METHOD StepDecoded : ZCore.ZString
VAR_INPUT
  stepIndex : INT;
END_VAR
VAR_INST
  _stepIndexDecoded : DrillingStep;
END_VAR
_stepIndexDecoded := stepIndex;
stepDecoded := TO_STRING(_stepIndexDecoded);
END_METHOD

END_FUNCTION_BLOCK

// ---- ZApp/Unit/Drilling/_States/DrillingSequenceAutomatic.TcPOU
FUNCTION_BLOCK DrillingSequenceAutomatic EXTENDS DrillingSequence IMPLEMENTS ZCore.ISequence
VAR
  _step : ZCore.Step(DrillingStep.AutomaticBegin, DrillingStep.AutomaticEnd);
END_VAR

IF NOT Busy THEN
  RETURN;
END_IF

IF OnStart(_step) THEN
  ; // init custom sequence variables here ...
END_IF

IF OnStop() THEN
  RETURN; // external stop was triggered
END_IF

IF OnHalt() THEN
  ; // Halting := TRUE; // Uncomment to acknowledge that the sequence is halting
END_IF

REPEAT
  LogStep();

  CASE _step.Index OF
    (* -------------------------------------------------------------------------------------------------------------------------------- *)
    DrillingStep.AutomaticBegin:
    (* -------------------------------------------------------------------------------------------------------------------------------- *)
      IF _step.OnEntry()
      THEN
        ;
      END_IF

      // Await(obj1:=, nextStep:=DrillingStep.AutomaticEnd);
      _step.SetNext(DrillingStep.AutomaticEnd);
    
    (* -------------------------------------------------------------------------------------------------------------------------------- *)
    DrillingStep.AutomaticEnd:
    (* -------------------------------------------------------------------------------------------------------------------------------- *)
      SetBusy(FALSE);
  
  ELSE
    Abort('sequence contains unhandled step');
  END_CASE
UNTIL _step.IsNotRepeatable() OR_ELSE NOT Busy END_REPEAT

END_FUNCTION_BLOCK

// ---- ZApp/Unit/Drilling/_States/DrillingSequenceStop.TcPOU
FUNCTION_BLOCK DrillingSequenceStop EXTENDS DrillingSequence IMPLEMENTS ZCore.ISequence
VAR
  _step : ZCore.Step(DrillingStep.StopBegin, DrillingStep.StopEnd);
  _timerSim : ZAux.Timer;
END_VAR

IF OnStart(_step) THEN
  ; // init custom sequence variables here ...
END_IF

REPEAT
  LogStep();

  CASE _step.Index OF
    (* -------------------------------------------------------------------------------------------------------------------------------- *)
    DrillingStep.StopBegin:
    (* -------------------------------------------------------------------------------------------------------------------------------- *)
      IF _step.OnEntry()
      THEN
        _timerSim.WaitAsync(5);
			END_IF
      
      Await(_timerSim, nextStep:=DrillingStep.StopEnd);
      // _step.SetNext(index:=DrillingStep.StopEnd);

    (* -------------------------------------------------------------------------------------------------------------------------------- *)
    DrillingStep.StopEnd:
    (* -------------------------------------------------------------------------------------------------------------------------------- *)    
      SetBusy(FALSE);
  
  ELSE
    Abort('sequence contains unhandled step');
  END_CASE
UNTIL _step.IsNotRepeatable() OR_ELSE NOT Busy END_REPEAT

END_FUNCTION_BLOCK

// ---- ZApp/Unit/Drilling/_States/DrillingSequenceGoHome.TcPOU
FUNCTION_BLOCK DrillingSequenceGoHome EXTENDS DrillingSequence IMPLEMENTS ZCore.ISequence
VAR
  _step : ZCore.Step(DrillingStep.GohomeBegin, DrillingStep.GohomeEnd);
  _timer : ZAux.Timer;
END_VAR

IF NOT Busy THEN
  RETURN;
END_IF

IF OnStart(_step) THEN
  ; // init custom sequence variables here ...
END_IF

IF OnStop() THEN
  RETURN; // external stop was triggered
END_IF

IF OnHalt() THEN
  ; // Halting := TRUE; // Uncomment to acknowledge that the sequence is halting
END_IF

REPEAT
  LogStep();

  CASE _step.Index OF
    (* -------------------------------------------------------------------------------------------------------------------------------- *)
    DrillingStep.GoHomeBegin:
    (* -------------------------------------------------------------------------------------------------------------------------------- *)
      IF _step.OnEntry()
      THEN
        _timer.WaitAsync(2);
			END_IF
      
      Await(_timer, nextStep:=DrillingStep.GoHomeEnd);
      // _step.SetNext(index:=DrillingStep.GoHomeEnd);

    (* -------------------------------------------------------------------------------------------------------------------------------- *)
    DrillingStep.GoHomeEnd:
    (* -------------------------------------------------------------------------------------------------------------------------------- *)
      SetBusy(FALSE);
  
  ELSE
    Abort('sequence contains unhandled step');
  END_CASE
UNTIL _step.IsNotRepeatable() OR_ELSE NOT Busy END_REPEAT

END_FUNCTION_BLOCK

// ---- ZApp/Unit/Drilling/_States/DrillingSequenceFaultReaction.TcPOU
FUNCTION_BLOCK DrillingSequenceFaultReaction EXTENDS DrillingSequence IMPLEMENTS ZCore.ISequence
VAR
  _step : ZCore.Step(DrillingStep.FaultReactionBegin, DrillingStep.FaultReactionEnd);
  _timerSim : ZAux.Timer;
END_VAR

IF OnStart(_step) THEN
  ; // init custom sequence variables here ...
END_IF

REPEAT
  LogStep();

  CASE _step.Index OF
    (* -------------------------------------------------------------------------------------------------------------------------------- *)
    DrillingStep.FaultReactionBegin:
    (* -------------------------------------------------------------------------------------------------------------------------------- *)
      IF _step.OnEntry()
      THEN
        _timerSim.WaitAsync(5);
			END_IF
      
      Await(_timerSim, nextStep:=DrillingStep.FaultReactionEnd);
      // _step.SetNext(index:=DrillingStep.FaultReactionEnd);

    (* -------------------------------------------------------------------------------------------------------------------------------- *)
    DrillingStep.FaultReactionEnd:
    (* -------------------------------------------------------------------------------------------------------------------------------- *)    
      SetBusy(FALSE);
  
  ELSE
    Abort('sequence contains unhandled step');
  END_CASE
UNTIL _step.IsNotRepeatable() OR_ELSE NOT Busy END_REPEAT

END_FUNCTION_BLOCK

// ---- ZApp/Unit/Assembly/AssemblyUnit.TcPOU
/// Declaration of a distinct unit of this application
FUNCTION_BLOCK AssemblyUnit EXTENDS ZApplication.Unit IMPLEMENTS IAssembly, ZAux.IStateMachineListener
VAR
  _equipment : AssemblyEquipment(THIS^);
  _data : AssemblyDataRef;
  _com : AssemblyComRef;

  _boot : AssemblySequenceBoot(THIS^);
  _automatic : AssemblySequenceAutomatic(THIS^);
  _stop : AssemblySequenceStop(THIS^);
  _gohome : AssemblySequenceGoHome(THIS^);
  _faultReaction : AssemblySequenceFaultReaction(THIS^);
  
  _statemachine : ZApplication.UnitStateMachine;

  _observeTimer : ZAux.Timer;
END_VAR

{attribute 'ZId' := '23221439-50f6-4bf8-9080-f9c9a764eb63'}

IF _observeTimer.Done THEN
  _observeTimer.WaitAsync(0.1);
  
  // monitor _com for requested actions (e.g. start homing, start automatic mode, ...)
  ObserveRequest(_com.Subscribe.Request.Start, ZApplication.UnitStateMachineState.Automatic);
  ObserveRequest(_com.Subscribe.Request.Stop, ZApplication.UnitStateMachineState.Stop);
  ObserveRequest(_com.Subscribe.Request.GoHome, ZApplication.UnitStateMachineState.GoHome);
  ObserveRequest(_com.Subscribe.Request.Halt, ZApplication.UnitStateMachineState.Halt);
  
  // provide relevant information via ADS
  _com.Publish.Request.Stop := _stateMachine.IsTransitionAllowed(ZApplication.UnitStateMachineState.Stop);
  _com.Publish.Request.Start := _stateMachine.IsTransitionAllowed(ZApplication.UnitStateMachineState.Automatic);
  _com.Publish.Request.GoHome := _stateMachine.IsTransitionAllowed(ZApplication.UnitStateMachineState.GoHome);
  _com.Publish.Request.Halt := _stateMachine.IsTransitionAllowed(ZApplication.UnitStateMachineState.Halt);

  _com.Publish.State := _stateMachine.State();
END_IF

METHOD FB_init : BOOL
VAR_INPUT
  bInitRetains : BOOL; // if TRUE, the retain variables are initialized (warm start / cold start)
  bInCopyCode : BOOL;  // if TRUE, the instance afterwards gets moved into the copy code (online change)
  parent : ZCore.IManagedObject; // caller of the Unit's cyclic method. If the Unit runs in its own context use 0
  name : ZCore.ZString;  // name of this unit as it should show up in the logger
  configdata : REFERENCE TO AssemblyDataConfig;  // reference to the configuration data that is used during boot to configure the Units equipment
  machinedata : REFERENCE TO AssemblyDataMachine; // reference to the machine data that is used through most sequences of the unit (motor speed, axes positions, ...)
  calibrationdata : REFERENCE TO AssemblyDataCalibration;  // reference to calibration that is determined by calibration sequences of the unit (static offsets, shifts)
  com : REFERENCE TO AssemblyCom;  // reference to the communication interface that is used to control this Unit via ADS
END_VAR
_name := name;

// initialize local logger decorator
_loggerDecorator.FB_init(bInitRetains, bInCopyCode, name, ZModuleProgram.Logger);
_alarmingDecorator.FB_init(bInitRetains, bInCopyCode, name, ZModuleProgram.Alarming);

// setup data
_data.Config REF= configdata;
_data.Machine REF= machinedata;
_data.Calibration REF= calibrationdata;
_com.Publish REF= com.Publish;
_com.Subscribe REF= com.Subscribe;

// ------- sequence initialization, map sequences of this unit to the statemachine -------
{attribute '__ZwPlcUnitInitSequenceImplementation__'} // Do not remove this attribute! It is used for code generation.
_statemachine.SetSequence(ZApplication.UnitStateMachineState.Boot, _boot);
_statemachine.SetSequence(ZApplication.UnitStateMachineState.FaultReaction, _faultReaction);
_statemachine.SetSequence(ZApplication.UnitStateMachineState.Gohome, _gohome);
_statemachine.SetSequence(ZApplication.UnitStateMachineState.Stop, _stop);
_statemachine.SetSequence(ZApplication.UnitStateMachineState.Automatic, _automatic);

_statemachine.SetName(_name);
_statemachine.SetListener(THIS^);
_statemachine.SetLogger(_logger);

// set initial state
_statemachine.SetState(ZApplication.UnitStateMachineState.Boot);
_statemachineIntrf := _statemachine;
END_METHOD

/// This method is called by a [Statemachine's startTransition method](xref:ZApplication.UnitStateMachine#startTransition)
/// if a given transition was failed (e.g. the transition is not allowed according to the state diagram of the state machine).
/// The State that was active previously in the StateMachine remains active and `requestedState` indicates which state transition
/// was requested by the user.
METHOD OnStartTransitionFailed
VAR_INPUT
  state : INT;  
  requestedState : INT;
END_VAR
END_METHOD

/// This method is called by a [Statemachine's startTransition method](xref:ZApplication.UnitStateMachine#startTransition)
/// if a given transition was successful. Please note, that at the time this event occurs, `state` still holds the
/// state that was active before calling `startTransition`, there is still one more call to this `state` to allow it to 
/// cleanup.
METHOD OnStartTransitionSucceeded
VAR_INPUT
  state : INT;  
  newState : INT;
END_VAR
END_METHOD

/// This method is called after a transition succeeded, right before the [start method of a sequence](xref:ZAux#start) is called.
/// The parameter `state` indicates the State that is active in the statemachine.
METHOD OnStateEntry
VAR_INPUT
  state : INT;
END_VAR
END_METHOD

/// This method is called after a sequence reported an error, but before the state machine starts its error handling.
METHOD OnStateError
VAR_INPUT
  state : INT;
END_VAR
END_METHOD

/// This method is called after a transition succeeded, right before the [stop method of a sequence](xref:ZAux#start) is called.
/// The parameter `state` indicates the State that is active in the statemachine.
METHOD OnStateExit
VAR_INPUT
  state : INT;  
END_VAR
END_METHOD

/// This method if a State has been executed successfully.
/// The parameter `state` indicates the State that is active in the statemachine.
METHOD OnStateSuccess
VAR_INPUT
  state : INT;    
END_VAR
END_METHOD

END_FUNCTION_BLOCK

// ---- ZApp/Unit/Assembly/_Equipment/AssemblyEquipment.TcPOU
/// This function block is a container for equipment that is used by this unit.
/// Equipment is grouped by its kind (actuator, axes, io, ...).
/// It extends from [ManagedObjectContainer](xref:ZCore.ManagedObjectContainer) such that the parent
/// (= the unit itself) can be passed to equipment instances.
FUNCTION_BLOCK AssemblyEquipment EXTENDS AssemblyContainer
VAR_INPUT
  Io : AssemblyIo(_parent);
  Actuator : AssemblyActuator(_parent);
  Axis : AssemblyAxis(_parent);
  Fieldbus : AssemblyFieldbus(_parent);
  Unit : AssemblyLinkedUnit(_parent);
END_VAR

END_FUNCTION_BLOCK

// ---- ZApp/Unit/Assembly/_SubObjects/AssemblyContainer.TcPOU
FUNCTION_BLOCK AssemblyContainer EXTENDS ZCore.ObjectContainer
VAR_INPUT
END_VAR
VAR_OUTPUT
END_VAR
VAR
  {attribute 'hide'}
  _parent : REFERENCE TO AssemblyUnit;
END_VAR

{ attribute 'hide' }
METHOD FB_init : BOOL
VAR_INPUT
	bInitRetains : BOOL; // if TRUE, the retain variables are initialized (warm start / cold start)
	bInCopyCode : BOOL;  // if TRUE, the instance afterwards gets moved into the copy code (online change)
  unit : REFERENCE TO AssemblyUnit;
END_VAR
_parent REF= unit;
END_METHOD

END_FUNCTION_BLOCK

// ---- ZApp/Unit/Assembly/_Equipment/AssemblyIo.TcPOU
/// This function block is a container for all I/Os that are used by this unit.
/// The parent of all objects can be directly transfered in their constructor (this is only relevant for equipment objects
/// that have to be managed (e.g. [DebouncedInput](xref:ZEquipment.DebouncedInput), [Light](xref:ZEquipment.Light), ...).
FUNCTION_BLOCK AssemblyIo EXTENDS AssemblyContainer
VAR
  {attribute 'hide'}
  _iobridge : ZApplication.IoBridge(_parent);
END_VAR
VAR_INPUT

{region "YellowLight : Light"}
  YellowLight : ZEquipment.Light(_parent);
  {attribute 'ZId' := 'd8b54b94-4c20-4805-9de3-a35aa5023c5d'}
{endregion}

{region "RedLight : Light"}
  RedLight : ZEquipment.Light(_parent);
  {attribute 'ZId' := '810dce14-d302-4e94-b60a-e39841040373'}
{endregion}

{region "GreenLight : Light"}
  GreenLight : ZEquipment.Light(_parent);
  {attribute 'ZId' := 'f5a46fca-074f-4557-8a14-cee504d2eb08'}
{endregion}

{region "PneumaticsOk : DigitalInput"}
  PneumaticsOk : ZEquipment.DigitalInput;
  {attribute 'ZId' := 'e461ecc5-0720-4dc8-ad47-eeb7ce01769f'}
{endregion}

{attribute '__ZwPlcUnitEquipmentDeclaration__'} // Do not remove this attribute! It is used for code generation.
END_VAR

IF _isInitialized
THEN
  RETURN;
END_IF

  _iobridge.SetLogger(_parent._logger);

{region "YellowLight : Light"}
  YellowLight.SetLogger(_parent._logger);
  YellowLight.SetName('YellowLight');
  YellowLight.SetSimulation(on:=_parent._data.Config.Simulated);
  YellowLight.SetLogic(ZEquipment.DigitalLogic.Normal);
  _ioBridge.AddLight(YellowLight, publish := _parent._com.Publish.Equipment.YellowLight, subscribe := _parent._com.Subscribe.Equipment.YellowLight);

  {region "UserInitCode"}
  // put your individual init code for this I/O here
  {endregion}

  {attribute 'ZId' := 'd8b54b94-4c20-4805-9de3-a35aa5023c5d'}
{endregion}

{region "RedLight : Light"}
  RedLight.SetLogger(_parent._logger);
  RedLight.SetName('RedLight');
  RedLight.SetSimulation(on:=_parent._data.Config.Simulated);
  RedLight.SetLogic(ZEquipment.DigitalLogic.Normal);
  _ioBridge.AddLight(RedLight, publish := _parent._com.Publish.Equipment.RedLight, subscribe := _parent._com.Subscribe.Equipment.RedLight);

  {region "UserInitCode"}
  // put your individual init code for this I/O here
  {endregion}

  {attribute 'ZId' := '810dce14-d302-4e94-b60a-e39841040373'}
{endregion}

{region "GreenLight : Light"}
  GreenLight.SetLogger(_parent._logger);
  GreenLight.SetName('GreenLight');
  GreenLight.SetSimulation(on:=_parent._data.Config.Simulated);
  GreenLight.SetLogic(ZEquipment.DigitalLogic.Normal);
  _ioBridge.AddLight(GreenLight, publish := _parent._com.Publish.Equipment.GreenLight, subscribe := _parent._com.Subscribe.Equipment.GreenLight);

  {region "UserInitCode"}
  // put your individual init code for this I/O here
  {endregion}

  {attribute 'ZId' := 'f5a46fca-074f-4557-8a14-cee504d2eb08'}
{endregion}

{region "PneumaticsOk : DigitalInput"}
  PneumaticsOk.SetLogger(_parent._logger);
  PneumaticsOk.SetName('PneumaticsOk');
  PneumaticsOk.SetSimulation(on:=_parent._data.Config.Simulated);
  PneumaticsOk.SetLogic(ZEquipment.DigitalLogic.Normal);
  _ioBridge.AddDigitalInput(PneumaticsOk, publish := _parent._com.Publish.Equipment.PneumaticsOk, subscribe := _parent._com.Subscribe.Equipment.PneumaticsOk);

  {region "UserInitCode"}
  // put your individual init code for this I/O here
  {endregion}

  {attribute 'ZId' := 'e461ecc5-0720-4dc8-ad47-eeb7ce01769f'}
{endregion}

{attribute '__ZwPlcUnitEquipmentImplementation__'} // Do not remove this attribute! It is used for code generation.

_isInitialized := TRUE;

END_FUNCTION_BLOCK

// ---- ZApp/Unit/Assembly/_Equipment/AssemblyActuator.TcPOU
/// This function block is a container for all actuator objects that are used by this unit.
/// The parent of all objects can be directly transfered in their constructor (this is only relevant for equipment objects
/// that have to be managed (e.g. [DebouncedInput](xref:ZEquipment.DebouncedInput), [Light](xref:ZEquipment.Light), ...).
FUNCTION_BLOCK AssemblyActuator EXTENDS AssemblyContainer
VAR
  {attribute 'hide'}
  _actuatorbridge : ZApplication.ActuatorBridge(_parent);
  {attribute 'hide'}
  _iobridge : ZApplication.IoBridge(_parent);
END_VAR
VAR_INPUT

{region "Horizontal : ActuatorDigitalBiLsPlusMinus"}
  Horizontal : AssemblyActuatorHorizontal(_parent);
  {attribute 'ZId' := 'bf04a1fd-9e2a-444c-be25-15a99c5011b8'}
{endregion}

{region "Gripper : ActuatorDigitalMonoPlusLsNo"}
  Gripper : AssemblyActuatorGripper(_parent);
  {attribute 'ZId' := 'd18888e4-9abb-463d-b01d-e5fd8694a677'}
{endregion}

{attribute '__ZwPlcUnitEquipmentDeclaration__'} // Do not remove this attribute! It is used for code generation.

  HorizontalListener : ActuatorHorizontalListener(Horizontal, _parent._equipment.Axis.Vertical, _parent._equipment.Io.YellowLight);
  HorizontalPneumaticsCheckListener : PneumaticsOkActuatorListener(Horizontal, _parent._equipment.Io.PneumaticsOk);
  
  GripperPneumaticsCheckListener : PneumaticsOkActuatorListener(Gripper, _parent._equipment.Io.PneumaticsOk);
END_VAR

IF _isInitialized
THEN
  RETURN;
END_IF

  _actuatorbridge.SetLogger(_parent._logger);

{region "Horizontal : ActuatorDigitalBiLsPlusMinus"}
  Horizontal.SetLogger(_parent._logger);
  Horizontal.SetName(name:='Horizontal', movePlusName:='ToTransport', moveMinusName:='ToAssembly', plusName:='AtTransport', minusName:='AtAssembly');
  Horizontal.SetSimulation(SEL(_parent._data.Config.Simulated, ActuatorDigitalSimulation.Disabled, ZEquipment.ActuatorDigitalSimulation.Automatic));
  Horizontal.SetSimulationUncertainty(uncertainty:=10);
  Horizontal.SetDelay(plusStartDuration:=0, plusEndDuration:=0, minusStartDuration:=0, minusEndDuration:=0, stop:=0);
  Horizontal.SetSwitchDuration(plusDuration:=0.2, minusDuration:=0.2);
  Horizontal.SetMovementDuration(plusDuration:=3, minusDuration:=3);
  Horizontal.SetTimeout(plusDuration:=5, minusDuration:=5);
  _actuatorbridge.AddActuatorDigital(Horizontal, publish := _parent._com.Publish.Equipment.Horizontal, subscribe := _parent._com.Subscribe.Equipment.Horizontal);
  _iobridge.AddDigitalOutput(Horizontal.MinusOutput, publish := _parent._com.Publish.Equipment.HorizontalToAssembly, subscribe := _parent._com.Subscribe.Equipment.HorizontalToAssembly);
  _iobridge.AddDigitalOutput(Horizontal.PlusOutput, publish := _parent._com.Publish.Equipment.HorizontalToTransport, subscribe := _parent._com.Subscribe.Equipment.HorizontalToTransport);
  _iobridge.AddDigitalInput(Horizontal.MinusInput, publish := _parent._com.Publish.Equipment.HorizontalAtAssembly, subscribe := _parent._com.Subscribe.Equipment.HorizontalAtAssembly);
  _iobridge.AddDigitalInput(Horizontal.PlusInput, publish := _parent._com.Publish.Equipment.HorizontalAtTransport, subscribe := _parent._com.Subscribe.Equipment.HorizontalAtTransport);
  {region "UserInitCode"}
  // put your individual init code for this Actuator here
  {endregion}

  {attribute 'ZId' := 'bf04a1fd-9e2a-444c-be25-15a99c5011b8'}
{endregion}

{region "Gripper : ActuatorDigitalMonoPlusLsNo"}
  Gripper.SetLogger(_parent._logger);
  Gripper.SetName(name:='Gripper', movePlusName:='Auf', moveMinusName:='Zu', plusName:='Offen', minusName:='Geschlossen');
  Gripper.SetSimulation(SEL(_parent._data.Config.Simulated, ActuatorDigitalSimulation.Disabled, ZEquipment.ActuatorDigitalSimulation.Automatic));
  Gripper.SetSimulationUncertainty(uncertainty:=10);
  Gripper.SetDelay(plusStartDuration:=0, plusEndDuration:=0, minusStartDuration:=0, minusEndDuration:=0, stop:=0);
  Gripper.SetSwitchDuration(plusDuration:=0, minusDuration:=0);
  Gripper.SetMovementDuration(plusDuration:=1, minusDuration:=1);
  Gripper.SetTimeout(plusDuration:=0, minusDuration:=0);
  _actuatorbridge.AddActuatorDigital(Gripper, publish := _parent._com.Publish.Equipment.Gripper, subscribe := _parent._com.Subscribe.Equipment.Gripper);
  _iobridge.AddDigitalOutput(Gripper.PlusOutput, publish := _parent._com.Publish.Equipment.GripperAuf, subscribe := _parent._com.Subscribe.Equipment.GripperAuf);
  {region "UserInitCode"}
  // put your individual init code for this Actuator here
  {endregion}

  {attribute 'ZId' := 'd18888e4-9abb-463d-b01d-e5fd8694a677'}
{endregion}

{attribute '__ZwPlcUnitEquipmentImplementation__'} // Do not remove this attribute! It is used for code generation.

  HorizontalListener.SetLogger(_parent._logger);
  HorizontalListener.SetName('HorizontalActuatorListener');
  
  HorizontalPneumaticsCheckListener.SetLogger(_parent._logger);
  HorizontalPneumaticsCheckListener.SetName('HorizontalPneumaticsCheckListener');
  HorizontalPneumaticsCheckListener.SetPneumaticsOkIo(_parent._equipment.Io.PneumaticsOk);
  
  GripperPneumaticsCheckListener.SetLogger(_parent._logger);
  GripperPneumaticsCheckListener.SetName('HorizontalPneumaticsCheckListener');
  GripperPneumaticsCheckListener.SetPneumaticsOkIo(_parent._equipment.Io.PneumaticsOk);  

_isInitialized := TRUE;

END_FUNCTION_BLOCK

// ---- ZApp/Unit/Assembly/_Equipment/AssemblyActuatorHorizontal.TcPOU
FUNCTION_BLOCK AssemblyActuatorHorizontal EXTENDS ZEquipment.ActuatorDigitalBiLsPlusMinus

METHOD PUBLIC AtAssembly : BOOL
VAR_INPUT
END_VAR
AtAssembly := IsAtMinus();
END_METHOD

METHOD PUBLIC AtTransport : BOOL
VAR_INPUT
END_VAR
AtTransport := IsAtPlus();
END_METHOD

METHOD PUBLIC ToAssemblyAsync
VAR_INPUT
  startToken : ZCore.IStartToken;
END_VAR
MoveMinusAsync(startToken:=startToken);
END_METHOD

METHOD PUBLIC ToTransportAsync
VAR_INPUT
  startToken : ZCore.IStartToken;
END_VAR
MovePlusAsync(startToken:=startToken);
END_METHOD

END_FUNCTION_BLOCK

// ---- ZApp/Unit/Assembly/_Equipment/AssemblyActuatorGripper.TcPOU
FUNCTION_BLOCK AssemblyActuatorGripper EXTENDS ZEquipment.ActuatorDigitalMonoPlusLsNo

METHOD PUBLIC AufAsync
VAR_INPUT
  startToken : ZCore.IStartToken;
END_VAR
MovePlusAsync(startToken:=startToken);
END_METHOD

METHOD PUBLIC Geschlossen : BOOL
VAR_INPUT
END_VAR
Geschlossen := IsAtMinus();
END_METHOD

METHOD PUBLIC Offen : BOOL
VAR_INPUT
END_VAR
Offen := IsAtPlus();
END_METHOD

METHOD PUBLIC ZuAsync
VAR_INPUT
  startToken : ZCore.IStartToken;
END_VAR
MoveMinusAsync(startToken:=startToken);
END_METHOD

END_FUNCTION_BLOCK

// ---- ZApp/Unit/Assembly/_Equipment/ActuatorHorizontalListener.TcPOU
FUNCTION_BLOCK ActuatorHorizontalListener EXTENDS ZEquipment.ActuatorDigitalMoveListenerSequence
VAR
  _timer : ZAux.Timer;
  _step : ZCore.Step(ActuatorHorizontalListenerStep.PreMoveStepBegin, ActuatorHorizontalListenerStep.PreMoveStepEnd);
  _yellowLight : ZEquipment.ILight;
  _axis : ZEquipment.IAxisFeedbackPosition;
END_VAR

CASE THIS^.Movement
OF
  (* ############################################################################## *)
  ZEquipment.ActuatorDigitalMoveListenerMovementType.PreMoveMinus,
  ZEquipment.ActuatorDigitalMoveListenerMovementType.PreMovePlus:
  (* ############################################################################## *)
    IF OnStart(_step)
    THEN
      ;
    END_IF
    
    REPEAT
      LogStep();
      
      CASE _step.Index OF
        (* -------------------------------------------------------------------------------------------------------------------------------- *)
        ActuatorHorizontalListenerStep.PreMoveStepBegin:
        (* -------------------------------------------------------------------------------------------------------------------------------- *)
          _step.SetNext(ActuatorHorizontalListenerStep.PreMoveStepStartLightBlinking);
    
        (* -------------------------------------------------------------------------------------------------------------------------------- *)
        ActuatorHorizontalListenerStep.PreMoveStepStartLightBlinking:
        (* -------------------------------------------------------------------------------------------------------------------------------- *)
          IF _step.OnEntry()
          THEN
            _logger.Info('Start Light Blinking');
            _yellowLight.Enable(characteristic:=LightCharacteristic.Isophase);
          END_IF
        
          _step.SetNext(ActuatorHorizontalListenerStep.PreMoveStepCheckAxisVerticalPosition);
        
        (* -------------------------------------------------------------------------------------------------------------------------------- *)
        ActuatorHorizontalListenerStep.PreMoveStepCheckAxisVerticalPosition:
        (* -------------------------------------------------------------------------------------------------------------------------------- *)
          IF _step.OnEntry()
          THEN
            _logger.Info('Check Axis Position');
            _timer.WaitAsync(duration:=1.5);
          END_IF
        
          // Check if axis is positioned greater than 5mm
          IF _axis.ActualPosition > 5.0
          THEN
            Abort('Cant Move Actuator, Axis at wrong position, collission may occur');
          ELSE
            Await(obj1:=_timer, nextStep:=ActuatorHorizontalListenerStep.PreMoveStepEnd);
          END_IF          
        
        (* -------------------------------------------------------------------------------------------------------------------------------- *)
        ActuatorHorizontalListenerStep.PreMoveStepEnd:
        (* -------------------------------------------------------------------------------------------------------------------------------- *)
          SetBusy(FALSE);
      
      ELSE
        Abort('sequence contains unhandled step');
      END_CASE
    UNTIL _step.IsNotRepeatable() OR_ELSE NOT Busy END_REPEAT
  
  (* ############################################################################## *)
  ZEquipment.ActuatorDigitalMoveListenerMovementType.PostMoveMinus,
  ZEquipment.ActuatorDigitalMoveListenerMovementType.PostMovePlus:
  (* ############################################################################## *)
    _yellowLight.Enable(characteristic:=LightCharacteristic.FixedOff);
    SetBusy(FALSE);
    
END_CASE

METHOD FB_init : BOOL
VAR_INPUT
 bInitRetains : BOOL;
 bInCopyCode : BOOL;
 actuator : REFERENCE TO ActuatorDigital;
 axis : ZEquipment.IAxisFeedbackPosition;
 light : ZEquipment.ILight;
END_VAR
_yellowLight := light;
_axis := axis;
END_METHOD

END_FUNCTION_BLOCK

// ---- ZApp/Unit/Assembly/_Equipment/PneumaticsOkActuatorListener.TcPOU
FUNCTION_BLOCK PneumaticsOkActuatorListener EXTENDS ZEquipment.ActuatorDigitalMoveListenerSequence
VAR
  _pneumaticsOk : ZEquipment.IDigital;
END_VAR

CASE THIS^.Movement
OF
  ZEquipment.ActuatorDigitalMoveListenerMovementType.PreMoveMinus,
  ZEquipment.ActuatorDigitalMoveListenerMovementType.PreMovePlus:
    // Checking if pneumatics are ok and if not abort actuator action
    IF _pneumaticsOk <> 0 AND_THEN NOT _pneumaticsOk.Enabled
    THEN
      Abort('Pneumatics are not OK; check pressure and try again!');
      RETURN;
		END_IF
    
  ZEquipment.ActuatorDigitalMoveListenerMovementType.PostMoveMinus,
  ZEquipment.ActuatorDigitalMoveListenerMovementType.PostMovePlus:
    ;
    
END_CASE

SetBusy(FALSE);

METHOD FB_init : BOOL
VAR_INPUT
 bInitRetains : BOOL;
 bInCopyCode : BOOL;
 actuator : REFERENCE TO ActuatorDigital;
 pneumaticsOk : ZEquipment.IDigital;
END_VAR
_pneumaticsOk := pneumaticsOk;
END_METHOD

METHOD SetPneumaticsOkIo
VAR_INPUT
  intrf : ZEquipment.IDigital;
END_VAR
_pneumaticsOk := intrf;
END_METHOD

END_FUNCTION_BLOCK

// ---- ZApp/Unit/Assembly/_Equipment/AssemblyAxis.TcPOU
/// This function block is a container for all axis objects that are used by this unit.
/// The parent of all objects can be directly transfered in their constructor (this is only relevant for equipment objects
/// that have to be managed (e.g. [DebouncedInput](xref:ZEquipment.DebouncedInput), [Light](xref:ZEquipment.Light), ...).
FUNCTION_BLOCK AssemblyAxis EXTENDS AssemblyContainer
VAR
  {attribute 'hide'}
  _axisbridge : ZApplication.AxisBridge(_parent);
END_VAR
VAR_INPUT

{region "Vertical : AxisPlcOpenMc"}
  Vertical : ZEquipment.AxisPlcOpenMc(_parent);
  {attribute 'ZId' := '59ce020b-a4f8-4d7a-a0dc-8b778ee4fde8'}
{endregion}

{attribute '__ZwPlcUnitEquipmentDeclaration__'} // Do not remove this attribute! It is used for code generation.
END_VAR

IF _isInitialized
THEN
  RETURN;
END_IF

  _axisbridge.SetLogger(_parent._logger);

{region "Vertical : AxisPlcOpenMc"}
  Vertical.SetLogger(_parent._logger);
  Vertical.SetName(name:='Vertical');
  Vertical.SetSimulation(_parent._data.Config.Simulated);
  _axisbridge.AddAxisPlcOpenMc(axis:=Vertical, publish:=_parent._com.Publish.Equipment.Vertical, subscribe:=_parent._com.Subscribe.Equipment.Vertical);

  {region "UserInitCode"}
  // put your individual init code for this Axis here
  {endregion}

  {attribute 'ZId' := '59ce020b-a4f8-4d7a-a0dc-8b778ee4fde8'}
{endregion}

{attribute '__ZwPlcUnitEquipmentImplementation__'} // Do not remove this attribute! It is used for code generation.

_isInitialized := TRUE;

END_FUNCTION_BLOCK

// ---- ZApp/Unit/Assembly/_Equipment/AssemblyFieldbus.TcPOU
/// This function block is a container for all axis objects that are used by this unit.
/// The parent of all objects can be directly transfered in their constructor (this is only relevant for equipment objects
/// that have to be managed (e.g. [DebouncedInput](xref:ZEquipment.DebouncedInput), [Light](xref:ZEquipment.Light), ...).
FUNCTION_BLOCK AssemblyFieldbus EXTENDS AssemblyContainer
VAR
END_VAR
VAR_INPUT

{attribute '__ZwPlcUnitEquipmentDeclaration__'} // Do not remove this attribute! It is used for code generation.
END_VAR

IF _isInitialized
THEN
  RETURN;
END_IF

{attribute '__ZwPlcUnitEquipmentImplementation__'} // Do not remove this attribute! It is used for code generation.

_isInitialized := TRUE;

END_FUNCTION_BLOCK

// ---- ZApp/Unit/Assembly/_Equipment/AssemblyLinkedUnit.TcPOU
/// This function block is a container for all linked units that are used by this unit.
/// Linked units can be addressed through their individual interface.
FUNCTION_BLOCK AssemblyLinkedUnit EXTENDS AssemblyContainer
VAR_INPUT

{attribute '__ZwPlcUnitEquipmentDeclaration__'} // Do not remove this attribute! It is used for code generation.
END_VAR

IF _isInitialized
THEN
  RETURN;
END_IF

{attribute '__ZwPlcUnitEquipmentImplementation__'} // Do not remove this attribute! It is used for code generation.

_isInitialized := TRUE;

END_FUNCTION_BLOCK

// ---- ZApp/Unit/Assembly/_States/AssemblySequenceBoot.TcPOU
FUNCTION_BLOCK AssemblySequenceBoot EXTENDS AssemblySequence IMPLEMENTS ZCore.ISequence
VAR
  _step : ZCore.Step(AssemblyStep.BootBegin, AssemblyStep.BootEnd);
END_VAR

IF OnStart(_step) THEN
  ; // init custom sequence variables here ...
END_IF

REPEAT
  LogStep();

  CASE _step.Index OF
    (* -------------------------------------------------------------------------------------------------------------------------------- *)
    AssemblyStep.BootBegin:
    (* -------------------------------------------------------------------------------------------------------------------------------- *)
      IF _step.OnEntry()
      THEN
        // initialize equipment
        _io();
        _actuator();
        _fieldbus();
        _axis();
        _unit();
      END_IF
      
      _parent._objectManager.Cyclic();      
      Assert(_parent._objectManager);
      IF _parent._objectManager.Done
      THEN
        _step.SetNext(AssemblyStep.BootSwitchOnPneumaticsOkInSimulation);
      END_IF

    (* -------------------------------------------------------------------------------------------------------------------------------- *)
    AssemblyStep.BootSwitchOnPneumaticsOkInSimulation:
    (* -------------------------------------------------------------------------------------------------------------------------------- *)
      IF _step.OnEntry()
      THEN        
        // This IO is an input so this line will only have some effect if PneumaticsOk is simulated to feedback a 
        // functioning pneumatics system to the application in simulation mode
        _io.PneumaticsOk.Enable(TRUE);
      END_IF
      
      _step.SetNext(index:=AssemblyStep.BootEnd);

    (* -------------------------------------------------------------------------------------------------------------------------------- *)
    AssemblyStep.BootEnd:
    (* -------------------------------------------------------------------------------------------------------------------------------- *)
      SetBusy(FALSE);
      
  ELSE
    Abort('sequence contains unhandled step');
  END_CASE
UNTIL _step.IsNotRepeatable() OR_ELSE NOT Busy END_REPEAT

END_FUNCTION_BLOCK

// ---- ZApp/Unit/Assembly/_SubObjects/AssemblySequence.TcPOU
FUNCTION_BLOCK AssemblySequence EXTENDS ZApplication.Sequence
VAR
  {attribute 'hide'}
  _parent : REFERENCE TO AssemblyUnit;
  _io : REFERENCE TO AssemblyIo;
  _actuator : REFERENCE TO AssemblyActuator;
  _fieldbus : REFERENCE TO AssemblyFieldbus;
  _axis : REFERENCE TO AssemblyAxis;
  _data : REFERENCE TO AssemblyDataRef;
  _unit : REFERENCE TO AssemblyLinkedUnit;  
END_VAR

METHOD FB_init : BOOL
VAR_INPUT
  bInitRetains : BOOL; // if TRUE, the retain variables are initialized (warm start / cold start)
  bInCopyCode : BOOL;  // if TRUE, the instance afterwards gets moved into the copy code (online change)
  unit : REFERENCE TO AssemblyUnit;
END_VAR
_parent REF= unit;
_alarming := unit._alarming;
_io REF= unit._equipment.Io;
_actuator REF= unit._equipment.Actuator;
_fieldbus REF= unit._equipment.Fieldbus;
_axis REF= unit._equipment.Axis;
_unit REF= unit._equipment.Unit;
_data REF= unit._data;
_loggerDiagnostics.SetLogger(unit._logger);
END_METHOD

METHOD StepDecoded : ZCore.ZString
VAR_INPUT
  stepIndex : INT;
END_VAR
VAR_INST
  _stepIndexDecoded : AssemblyStep;
END_VAR
_stepIndexDecoded := stepIndex;
stepDecoded := TO_STRING(_stepIndexDecoded);
END_METHOD

END_FUNCTION_BLOCK

// ---- ZApp/Unit/Assembly/_States/AssemblySequenceAutomatic.TcPOU
FUNCTION_BLOCK AssemblySequenceAutomatic EXTENDS AssemblySequence IMPLEMENTS ZCore.ISequence
VAR
  _step : ZCore.Step(AssemblyStep.AutomaticBegin, AssemblyStep.AutomaticEnd);
END_VAR

IF NOT Busy THEN
  RETURN;
END_IF

IF OnStart(_step) THEN
  ; // init custom sequence variables here ...
END_IF

IF OnStop() THEN
  RETURN; // external stop was triggered
END_IF

IF OnHalt() THEN
  ; // Halting := TRUE; // Uncomment to acknowledge that the sequence is halting
END_IF

REPEAT
  LogStep();

  CASE _step.Index OF
    (* -------------------------------------------------------------------------------------------------------------------------------- *)
    AssemblyStep.AutomaticBegin:
    (* -------------------------------------------------------------------------------------------------------------------------------- *)
      IF _step.OnEntry()
      THEN
        ;
      END_IF

      // Await(obj1:=, nextStep:=AssemblyStep.AutomaticEnd);
      _step.SetNext(AssemblyStep.AutomaticEnd);
    
    (* -------------------------------------------------------------------------------------------------------------------------------- *)
    AssemblyStep.AutomaticEnd:
    (* -------------------------------------------------------------------------------------------------------------------------------- *)
      SetBusy(FALSE);
  
  ELSE
    Abort('sequence contains unhandled step');
  END_CASE
UNTIL _step.IsNotRepeatable() OR_ELSE NOT Busy END_REPEAT

END_FUNCTION_BLOCK

// ---- ZApp/Unit/Assembly/_States/AssemblySequenceStop.TcPOU
FUNCTION_BLOCK AssemblySequenceStop EXTENDS AssemblySequence IMPLEMENTS ZCore.ISequence
VAR
  _step : ZCore.Step(AssemblyStep.StopBegin, AssemblyStep.StopEnd);
  _timerSim : ZAux.Timer;
END_VAR

IF OnStart(_step) THEN
  ; // init custom sequence variables here ...
END_IF

REPEAT
  LogStep();

  CASE _step.Index OF
    (* -------------------------------------------------------------------------------------------------------------------------------- *)
    AssemblyStep.StopBegin:
    (* -------------------------------------------------------------------------------------------------------------------------------- *)
      IF _step.OnEntry()
      THEN
        _timerSim.WaitAsync(5);
			END_IF
      
      Await(_timerSim, nextStep:=AssemblyStep.StopEnd);
      // _step.SetNext(index:=AssemblyStep.StopEnd);

    (* -------------------------------------------------------------------------------------------------------------------------------- *)
    AssemblyStep.StopEnd:
    (* -------------------------------------------------------------------------------------------------------------------------------- *)    
      SetBusy(FALSE);
  
  ELSE
    Abort('sequence contains unhandled step');
  END_CASE
UNTIL _step.IsNotRepeatable() OR_ELSE NOT Busy END_REPEAT

END_FUNCTION_BLOCK

// ---- ZApp/Unit/Assembly/_States/AssemblySequenceGoHome.TcPOU
FUNCTION_BLOCK AssemblySequenceGoHome EXTENDS AssemblySequence IMPLEMENTS ZCore.ISequence
VAR
  _step : ZCore.Step(AssemblyStep.GohomeBegin, AssemblyStep.GohomeEnd);
  _timer : ZAux.Timer;
END_VAR

IF NOT Busy THEN
  RETURN;
END_IF

IF OnStart(_step) THEN
  ; // init custom sequence variables here ...
END_IF

IF OnStop() THEN
  RETURN; // external stop was triggered
END_IF

IF OnHalt() THEN
  ; // Halting := TRUE; // Uncomment to acknowledge that the sequence is halting
END_IF

REPEAT
  LogStep();

  CASE _step.Index OF
    (* -------------------------------------------------------------------------------------------------------------------------------- *)
    AssemblyStep.GoHomeBegin:
    (* -------------------------------------------------------------------------------------------------------------------------------- *)
      IF _step.OnEntry()
      THEN
        _timer.WaitAsync(2);
			END_IF
      
      Await(_timer, nextStep:=AssemblyStep.GoHomeGoToHomePos);
      // _step.SetNext(index:=AssemblyStep.GoHomeEnd);

    (* -------------------------------------------------------------------------------------------------------------------------------- *)
    AssemblyStep.GoHomeGoToHomePos:
    (* -------------------------------------------------------------------------------------------------------------------------------- *)
      IF _step.OnEntry()
      THEN        
        _axis.Vertical.MoveAbsoluteAsync(THIS^, 10.0, 2.0);
      END_IF
      
      Await(obj1:=_axis.Vertical, nextStep:=AssemblyStep.GoHomeEnd);

    (* -------------------------------------------------------------------------------------------------------------------------------- *)
    AssemblyStep.GoHomeEnd:
    (* -------------------------------------------------------------------------------------------------------------------------------- *)
      SetBusy(FALSE);
  
  ELSE
    Abort('sequence contains unhandled step');
  END_CASE
UNTIL _step.IsNotRepeatable() OR_ELSE NOT Busy END_REPEAT

END_FUNCTION_BLOCK

// ---- ZApp/Unit/Assembly/_States/AssemblySequenceFaultReaction.TcPOU
FUNCTION_BLOCK AssemblySequenceFaultReaction EXTENDS AssemblySequence IMPLEMENTS ZCore.ISequence
VAR
  _step : ZCore.Step(AssemblyStep.FaultReactionBegin, AssemblyStep.FaultReactionEnd);
  _timerSim : ZAux.Timer;
END_VAR

IF OnStart(_step) THEN
  ; // init custom sequence variables here ...
END_IF

REPEAT
  LogStep();

  CASE _step.Index OF
    (* -------------------------------------------------------------------------------------------------------------------------------- *)
    AssemblyStep.FaultReactionBegin:
    (* -------------------------------------------------------------------------------------------------------------------------------- *)
      IF _step.OnEntry()
      THEN
        _timerSim.WaitAsync(5);
			END_IF
      
      Await(_timerSim, nextStep:=AssemblyStep.FaultReactionEnd);
      // _step.SetNext(index:=AssemblyStep.FaultReactionEnd);

    (* -------------------------------------------------------------------------------------------------------------------------------- *)
    AssemblyStep.FaultReactionEnd:
    (* -------------------------------------------------------------------------------------------------------------------------------- *)    
      SetBusy(FALSE);
  
  ELSE
    Abort('sequence contains unhandled step');
  END_CASE
UNTIL _step.IsNotRepeatable() OR_ELSE NOT Busy END_REPEAT

END_FUNCTION_BLOCK

// ---- ZApp/Unit/QualityInspection/QualityInspectionUnit.TcPOU
/// Declaration of a distinct unit of this application
FUNCTION_BLOCK QualityInspectionUnit EXTENDS ZApplication.Unit IMPLEMENTS IQualityInspection, ZAux.IStateMachineListener
VAR
  _equipment : QualityInspectionEquipment(THIS^);
  _data : QualityInspectionDataRef;
  _com : QualityInspectionComRef;

  _boot : QualityInspectionSequenceBoot(THIS^);
  _automatic : QualityInspectionSequenceAutomatic(THIS^);
  _stop : QualityInspectionSequenceStop(THIS^);
  _gohome : QualityInspectionSequenceGoHome(THIS^);
  _faultReaction : QualityInspectionSequenceFaultReaction(THIS^);
  
  _statemachine : ZApplication.UnitStateMachine;

  _observeTimer : ZAux.Timer;
END_VAR

{attribute 'ZId' := '97aa7849-00c7-453f-b185-2784616f7454'}

IF _observeTimer.Done THEN
  _observeTimer.WaitAsync(0.1);
  
  // monitor _com for requested actions (e.g. start homing, start automatic mode, ...)
  ObserveRequest(_com.Subscribe.Request.Start, ZApplication.UnitStateMachineState.Automatic);
  ObserveRequest(_com.Subscribe.Request.Stop, ZApplication.UnitStateMachineState.Stop);
  ObserveRequest(_com.Subscribe.Request.GoHome, ZApplication.UnitStateMachineState.GoHome);
  ObserveRequest(_com.Subscribe.Request.Halt, ZApplication.UnitStateMachineState.Halt);
  
  // provide relevant information via ADS
  _com.Publish.Request.Stop := _stateMachine.IsTransitionAllowed(ZApplication.UnitStateMachineState.Stop);
  _com.Publish.Request.Start := _stateMachine.IsTransitionAllowed(ZApplication.UnitStateMachineState.Automatic);
  _com.Publish.Request.GoHome := _stateMachine.IsTransitionAllowed(ZApplication.UnitStateMachineState.GoHome);
  _com.Publish.Request.Halt := _stateMachine.IsTransitionAllowed(ZApplication.UnitStateMachineState.Halt);

  _com.Publish.State := _stateMachine.State();
END_IF

METHOD FB_init : BOOL
VAR_INPUT
  bInitRetains : BOOL; // if TRUE, the retain variables are initialized (warm start / cold start)
  bInCopyCode : BOOL;  // if TRUE, the instance afterwards gets moved into the copy code (online change)
  parent : ZCore.IManagedObject; // caller of the Unit's cyclic method. If the Unit runs in its own context use 0
  name : ZCore.ZString;  // name of this unit as it should show up in the logger
  configdata : REFERENCE TO QualityInspectionDataConfig;  // reference to the configuration data that is used during boot to configure the Units equipment
  machinedata : REFERENCE TO QualityInspectionDataMachine; // reference to the machine data that is used through most sequences of the unit (motor speed, axes positions, ...)
  calibrationdata : REFERENCE TO QualityInspectionDataCalibration;  // reference to calibration that is determined by calibration sequences of the unit (static offsets, shifts)
  com : REFERENCE TO QualityInspectionCom;  // reference to the communication interface that is used to control this Unit via ADS
END_VAR
_name := name;

// initialize local logger decorator
_loggerDecorator.FB_init(bInitRetains, bInCopyCode, name, ZModuleProgram.Logger);
_alarmingDecorator.FB_init(bInitRetains, bInCopyCode, name, ZModuleProgram.Alarming);

// setup data
_data.Config REF= configdata;
_data.Machine REF= machinedata;
_data.Calibration REF= calibrationdata;
_com.Publish REF= com.Publish;
_com.Subscribe REF= com.Subscribe;

// ------- sequence initialization, map sequences of this unit to the statemachine -------
{attribute '__ZwPlcUnitInitSequenceImplementation__'} // Do not remove this attribute! It is used for code generation.
_statemachine.SetSequence(ZApplication.UnitStateMachineState.Boot, _boot);
_statemachine.SetSequence(ZApplication.UnitStateMachineState.FaultReaction, _faultReaction);
_statemachine.SetSequence(ZApplication.UnitStateMachineState.Gohome, _gohome);
_statemachine.SetSequence(ZApplication.UnitStateMachineState.Stop, _stop);
_statemachine.SetSequence(ZApplication.UnitStateMachineState.Automatic, _automatic);

_statemachine.SetName(_name);
_statemachine.SetListener(THIS^);
_statemachine.SetLogger(_logger);

// set initial state
_statemachine.SetState(ZApplication.UnitStateMachineState.Boot);
_statemachineIntrf := _statemachine;
END_METHOD

/// This method is called by a [Statemachine's startTransition method](xref:ZApplication.UnitStateMachine#startTransition)
/// if a given transition was failed (e.g. the transition is not allowed according to the state diagram of the state machine).
/// The State that was active previously in the StateMachine remains active and `requestedState` indicates which state transition
/// was requested by the user.
METHOD OnStartTransitionFailed
VAR_INPUT
  state : INT;  
  requestedState : INT;
END_VAR
END_METHOD

/// This method is called by a [Statemachine's startTransition method](xref:ZApplication.UnitStateMachine#startTransition)
/// if a given transition was successful. Please note, that at the time this event occurs, `state` still holds the
/// state that was active before calling `startTransition`, there is still one more call to this `state` to allow it to 
/// cleanup.
METHOD OnStartTransitionSucceeded
VAR_INPUT
  state : INT;  
  newState : INT;
END_VAR
END_METHOD

/// This method is called after a transition succeeded, right before the [start method of a sequence](xref:ZAux#start) is called.
/// The parameter `state` indicates the State that is active in the statemachine.
METHOD OnStateEntry
VAR_INPUT
  state : INT;
END_VAR
END_METHOD

/// This method is called after a sequence reported an error, but before the state machine starts its error handling.
METHOD OnStateError
VAR_INPUT
  state : INT;
END_VAR
END_METHOD

/// This method is called after a transition succeeded, right before the [stop method of a sequence](xref:ZAux#start) is called.
/// The parameter `state` indicates the State that is active in the statemachine.
METHOD OnStateExit
VAR_INPUT
  state : INT;  
END_VAR
END_METHOD

/// This method if a State has been executed successfully.
/// The parameter `state` indicates the State that is active in the statemachine.
METHOD OnStateSuccess
VAR_INPUT
  state : INT;    
END_VAR
END_METHOD

END_FUNCTION_BLOCK

// ---- ZApp/Unit/QualityInspection/_Equipment/QualityInspectionEquipment.TcPOU
/// This function block is a container for equipment that is used by this unit.
/// Equipment is grouped by its kind (actuator, axes, io, ...).
/// It extends from [ManagedObjectContainer](xref:ZCore.ManagedObjectContainer) such that the parent
/// (= the unit itself) can be passed to equipment instances.
FUNCTION_BLOCK QualityInspectionEquipment EXTENDS QualityInspectionContainer
VAR_INPUT
  Io : QualityInspectionIo(_parent);
  Actuator : QualityInspectionActuator(_parent);
  Axis : QualityInspectionAxis(_parent);
  Fieldbus : QualityInspectionFieldbus(_parent);
  Unit : QualityInspectionLinkedUnit(_parent);
END_VAR

END_FUNCTION_BLOCK

// ---- ZApp/Unit/QualityInspection/_SubObjects/QualityInspectionContainer.TcPOU
FUNCTION_BLOCK QualityInspectionContainer EXTENDS ZCore.ObjectContainer
VAR_INPUT
END_VAR
VAR_OUTPUT
END_VAR
VAR
  {attribute 'hide'}
  _parent : REFERENCE TO QualityInspectionUnit;
END_VAR

{ attribute 'hide' }
METHOD FB_init : BOOL
VAR_INPUT
	bInitRetains : BOOL; // if TRUE, the retain variables are initialized (warm start / cold start)
	bInCopyCode : BOOL;  // if TRUE, the instance afterwards gets moved into the copy code (online change)
  unit : REFERENCE TO QualityInspectionUnit;
END_VAR
_parent REF= unit;
END_METHOD

END_FUNCTION_BLOCK

// ---- ZApp/Unit/QualityInspection/_Equipment/QualityInspectionIo.TcPOU
/// This function block is a container for all I/Os that are used by this unit.
/// The parent of all objects can be directly transfered in their constructor (this is only relevant for equipment objects
/// that have to be managed (e.g. [DebouncedInput](xref:ZEquipment.DebouncedInput), [Light](xref:ZEquipment.Light), ...).
FUNCTION_BLOCK QualityInspectionIo EXTENDS QualityInspectionContainer
VAR
  {attribute 'hide'}
  _iobridge : ZApplication.IoBridge(_parent);
END_VAR
VAR_INPUT

{region "TriggerCam : PulsedOutput"}
  TriggerCam : ZEquipment.ImpulseOutput(_parent);
  {attribute 'ZId' := 'c63d51c9-4589-40b4-ac78-45c3ff2f3b57'}
{endregion}

{region "EnableLight : DigitalOutput"}
  EnableLight : ZEquipment.DigitalOutput;
  {attribute 'ZId' := '57b0de1b-3452-4c6c-9481-eeca6b7d3a02'}
{endregion}

{region "CamOk : DigitalInput"}
  CamOk : ZEquipment.DigitalInput;
  {attribute 'ZId' := '27a646f9-ab74-4898-af0f-5400552173e7'}
{endregion}

{attribute '__ZwPlcUnitEquipmentDeclaration__'} // Do not remove this attribute! It is used for code generation.
END_VAR

IF _isInitialized
THEN
  RETURN;
END_IF

  _iobridge.SetLogger(_parent._logger);

{region "TriggerCam : PulsedOutput"}
  TriggerCam.SetLogger(0);
  TriggerCam.SetName('TriggerCam');
  TriggerCam.SetSimulation(on:=_parent._data.Config.Simulated);
  TriggerCam.SetLogic(ZEquipment.DigitalLogic.Normal);
  _ioBridge.AddImpulseOutput(TriggerCam, publish := _parent._com.Publish.Equipment.TriggerCam, subscribe := _parent._com.Subscribe.Equipment.TriggerCam);

  {region "UserInitCode"}
  // put your individual init code for this I/O here
  {endregion}

  {attribute 'ZId' := 'c63d51c9-4589-40b4-ac78-45c3ff2f3b57'}
{endregion}

{region "EnableLight : DigitalOutput"}
  EnableLight.SetLogger(_parent._logger);
  EnableLight.SetName('EnableLight');
  EnableLight.SetSimulation(on:=_parent._data.Config.Simulated);
  EnableLight.SetLogic(ZEquipment.DigitalLogic.Normal);
  _ioBridge.AddDigitalOutput(EnableLight, publish := _parent._com.Publish.Equipment.EnableLight, subscribe := _parent._com.Subscribe.Equipment.EnableLight);

  {region "UserInitCode"}
  // put your individual init code for this I/O here
  {endregion}

  {attribute 'ZId' := '57b0de1b-3452-4c6c-9481-eeca6b7d3a02'}
{endregion}

{region "CamOk : DigitalInput"}
  CamOk.SetLogger(_parent._logger);
  CamOk.SetName('CamOk');
  CamOk.SetSimulation(on:=_parent._data.Config.Simulated);
  CamOk.SetLogic(ZEquipment.DigitalLogic.Normal);
  _ioBridge.AddDigitalInput(CamOk, publish := _parent._com.Publish.Equipment.CamOk, subscribe := _parent._com.Subscribe.Equipment.CamOk);

  {region "UserInitCode"}
  // put your individual init code for this I/O here
  {endregion}

  {attribute 'ZId' := '27a646f9-ab74-4898-af0f-5400552173e7'}
{endregion}

{attribute '__ZwPlcUnitEquipmentImplementation__'} // Do not remove this attribute! It is used for code generation.

_isInitialized := TRUE;

END_FUNCTION_BLOCK

// ---- ZApp/Unit/QualityInspection/_Equipment/QualityInspectionActuator.TcPOU
/// This function block is a container for all actuator objects that are used by this unit.
/// The parent of all objects can be directly transfered in their constructor (this is only relevant for equipment objects
/// that have to be managed (e.g. [DebouncedInput](xref:ZEquipment.DebouncedInput), [Light](xref:ZEquipment.Light), ...).
FUNCTION_BLOCK QualityInspectionActuator EXTENDS QualityInspectionContainer
VAR
  {attribute 'hide'}
  _actuatorbridge : ZApplication.ActuatorBridge(_parent);
  {attribute 'hide'}
  _iobridge : ZApplication.IoBridge(_parent);
END_VAR
VAR_INPUT

{attribute '__ZwPlcUnitEquipmentDeclaration__'} // Do not remove this attribute! It is used for code generation.
END_VAR

IF _isInitialized
THEN
  RETURN;
END_IF

  _actuatorbridge.SetLogger(_parent._logger);

{attribute '__ZwPlcUnitEquipmentImplementation__'} // Do not remove this attribute! It is used for code generation.

_isInitialized := TRUE;

END_FUNCTION_BLOCK

// ---- ZApp/Unit/QualityInspection/_Equipment/QualityInspectionAxis.TcPOU
/// This function block is a container for all axis objects that are used by this unit.
/// The parent of all objects can be directly transfered in their constructor (this is only relevant for equipment objects
/// that have to be managed (e.g. [DebouncedInput](xref:ZEquipment.DebouncedInput), [Light](xref:ZEquipment.Light), ...).
FUNCTION_BLOCK QualityInspectionAxis EXTENDS QualityInspectionContainer
VAR
  {attribute 'hide'}
  _axisbridge : ZApplication.AxisBridge(_parent);
END_VAR
VAR_INPUT

{attribute '__ZwPlcUnitEquipmentDeclaration__'} // Do not remove this attribute! It is used for code generation.
END_VAR

IF _isInitialized
THEN
  RETURN;
END_IF

  _axisbridge.SetLogger(_parent._logger);

{attribute '__ZwPlcUnitEquipmentImplementation__'} // Do not remove this attribute! It is used for code generation.

_isInitialized := TRUE;

END_FUNCTION_BLOCK

// ---- ZApp/Unit/QualityInspection/_Equipment/QualityInspectionFieldbus.TcPOU
/// This function block is a container for all axis objects that are used by this unit.
/// The parent of all objects can be directly transfered in their constructor (this is only relevant for equipment objects
/// that have to be managed (e.g. [DebouncedInput](xref:ZEquipment.DebouncedInput), [Light](xref:ZEquipment.Light), ...).
FUNCTION_BLOCK QualityInspectionFieldbus EXTENDS QualityInspectionContainer
VAR
END_VAR
VAR_INPUT

{attribute '__ZwPlcUnitEquipmentDeclaration__'} // Do not remove this attribute! It is used for code generation.
END_VAR

IF _isInitialized
THEN
  RETURN;
END_IF

{attribute '__ZwPlcUnitEquipmentImplementation__'} // Do not remove this attribute! It is used for code generation.

_isInitialized := TRUE;

END_FUNCTION_BLOCK

// ---- ZApp/Unit/QualityInspection/_Equipment/QualityInspectionLinkedUnit.TcPOU
/// This function block is a container for all linked units that are used by this unit.
/// Linked units can be addressed through their individual interface.
FUNCTION_BLOCK QualityInspectionLinkedUnit EXTENDS QualityInspectionContainer
VAR_INPUT

{attribute '__ZwPlcUnitEquipmentDeclaration__'} // Do not remove this attribute! It is used for code generation.
END_VAR

IF _isInitialized
THEN
  RETURN;
END_IF

{attribute '__ZwPlcUnitEquipmentImplementation__'} // Do not remove this attribute! It is used for code generation.

_isInitialized := TRUE;

END_FUNCTION_BLOCK

// ---- ZApp/Unit/QualityInspection/_States/QualityInspectionSequenceBoot.TcPOU
FUNCTION_BLOCK QualityInspectionSequenceBoot EXTENDS QualityInspectionSequence IMPLEMENTS ZCore.ISequence
VAR
  _step : ZCore.Step(QualityInspectionStep.BootBegin, QualityInspectionStep.BootEnd);
END_VAR

IF OnStart(_step) THEN
  ; // init custom sequence variables here ...
END_IF

REPEAT
  LogStep();

  CASE _step.Index OF
    (* -------------------------------------------------------------------------------------------------------------------------------- *)
    QualityInspectionStep.BootBegin:
    (* -------------------------------------------------------------------------------------------------------------------------------- *)
      IF _step.OnEntry()
      THEN
        // initialize equipment
        _io();
        _actuator();
        _fieldbus();
        _axis();
        _unit();
      END_IF
      
      _parent._objectManager.Cyclic();      
      Assert(_parent._objectManager);
      IF _parent._objectManager.Done
      THEN
        _step.SetNext(QualityInspectionStep.BootEnd);
      END_IF

    (* -------------------------------------------------------------------------------------------------------------------------------- *)
    QualityInspectionStep.BootEnd:
    (* -------------------------------------------------------------------------------------------------------------------------------- *)
      SetBusy(FALSE);
      
  ELSE
    Abort('sequence contains unhandled step');
  END_CASE
UNTIL _step.IsNotRepeatable() OR_ELSE NOT Busy END_REPEAT

END_FUNCTION_BLOCK

// ---- ZApp/Unit/QualityInspection/_SubObjects/QualityInspectionSequence.TcPOU
FUNCTION_BLOCK QualityInspectionSequence EXTENDS ZApplication.Sequence
VAR
  {attribute 'hide'}
  _parent : REFERENCE TO QualityInspectionUnit;
  _io : REFERENCE TO QualityInspectionIo;
  _actuator : REFERENCE TO QualityInspectionActuator;
  _fieldbus : REFERENCE TO QualityInspectionFieldbus;
  _axis : REFERENCE TO QualityInspectionAxis;
  _data : REFERENCE TO QualityInspectionDataRef;
  _unit : REFERENCE TO QualityInspectionLinkedUnit;  
END_VAR

METHOD FB_init : BOOL
VAR_INPUT
  bInitRetains : BOOL; // if TRUE, the retain variables are initialized (warm start / cold start)
  bInCopyCode : BOOL;  // if TRUE, the instance afterwards gets moved into the copy code (online change)
  unit : REFERENCE TO QualityInspectionUnit;
END_VAR
_parent REF= unit;
_alarming := unit._alarming;
_io REF= unit._equipment.Io;
_actuator REF= unit._equipment.Actuator;
_fieldbus REF= unit._equipment.Fieldbus;
_axis REF= unit._equipment.Axis;
_unit REF= unit._equipment.Unit;
_data REF= unit._data;
_loggerDiagnostics.SetLogger(unit._logger);
END_METHOD

METHOD StepDecoded : ZCore.ZString
VAR_INPUT
  stepIndex : INT;
END_VAR
VAR_INST
  _stepIndexDecoded : QualityInspectionStep;
END_VAR
_stepIndexDecoded := stepIndex;
stepDecoded := TO_STRING(_stepIndexDecoded);
END_METHOD

END_FUNCTION_BLOCK

// ---- ZApp/Unit/QualityInspection/_States/QualityInspectionSequenceAutomatic.TcPOU
FUNCTION_BLOCK QualityInspectionSequenceAutomatic EXTENDS QualityInspectionSequence IMPLEMENTS ZCore.ISequence
VAR
  _step : ZCore.Step(QualityInspectionStep.AutomaticBegin, QualityInspectionStep.AutomaticEnd);
  _timer : ZAux.Timer;
  _simTimer : ZAux.Timer;
END_VAR

IF NOT Busy THEN
  RETURN;
END_IF

IF OnStart(_step) THEN
  ; // init custom sequence variables here ...
END_IF

IF OnStop() THEN
  RETURN; // external stop was triggered
END_IF

IF OnHalt() THEN
  ; // Halting := TRUE; // Uncomment to acknowledge that the sequence is halting
END_IF

REPEAT
  LogStep();

  CASE _step.Index OF
    (* -------------------------------------------------------------------------------------------------------------------------------- *)
    QualityInspectionStep.AutomaticBegin:
    (* -------------------------------------------------------------------------------------------------------------------------------- *)
      IF _step.OnEntry()
      THEN
        _timer.WaitAsync(1.0);
      END_IF

      _step.SetNext(QualityInspectionStep.AutomaticEnableLight);

    (* -------------------------------------------------------------------------------------------------------------------------------- *)
    QualityInspectionStep.AutomaticEnableLight:
    (* -------------------------------------------------------------------------------------------------------------------------------- *)
      IF _step.OnEntry()
      THEN        
        _io.EnableLight.Enable(TRUE);
      END_IF
      
      _step.SetNext(index:=QualityInspectionStep.AutomaticTriggerCam);

    (* -------------------------------------------------------------------------------------------------------------------------------- *)
    QualityInspectionStep.AutomaticTriggerCam:
    (* -------------------------------------------------------------------------------------------------------------------------------- *)
      IF _step.OnEntry()
      THEN        
        _io.TriggerCam.Duration := 0.5;
        _io.TriggerCam.RunAsync(startToken:=THIS^);
      END_IF
      
      Await(obj1:=_io.TriggerCam, nextStep:=QualityInspectionStep.AutomaticWaitTillCamSendsOk);

    (* -------------------------------------------------------------------------------------------------------------------------------- *)
    QualityInspectionStep.AutomaticWaitTillCamSendsOk:
    (* -------------------------------------------------------------------------------------------------------------------------------- *)
      IF _step.OnEntry()
      THEN        
        _simTimer.WaitAsync(1.5);
      END_IF
      
      IF _simTimer.Done
      THEN
        _io.CamOk.Enable(TRUE);
			END_IF
      
      IF _io.CamOk.RisingTrigger()
      THEN
        _io.CamOk.Enable(FALSE);
        _step.SetNext(index:=QualityInspectionStep.AutomaticEnd);
      END_IF
    
    (* -------------------------------------------------------------------------------------------------------------------------------- *)
    QualityInspectionStep.AutomaticEnd:
    (* -------------------------------------------------------------------------------------------------------------------------------- *)
      SetBusy(FALSE);
  
  ELSE
    Abort('sequence contains unhandled step');
  END_CASE
UNTIL _step.IsNotRepeatable() OR_ELSE NOT Busy END_REPEAT

END_FUNCTION_BLOCK

// ---- ZApp/Unit/QualityInspection/_States/QualityInspectionSequenceStop.TcPOU
FUNCTION_BLOCK QualityInspectionSequenceStop EXTENDS QualityInspectionSequence IMPLEMENTS ZCore.ISequence
VAR
  _step : ZCore.Step(QualityInspectionStep.StopBegin, QualityInspectionStep.StopEnd);
  _timerSim : ZAux.Timer;
END_VAR

IF OnStart(_step) THEN
  ; // init custom sequence variables here ...
END_IF

REPEAT
  LogStep();

  CASE _step.Index OF
    (* -------------------------------------------------------------------------------------------------------------------------------- *)
    QualityInspectionStep.StopBegin:
    (* -------------------------------------------------------------------------------------------------------------------------------- *)
      IF _step.OnEntry()
      THEN
        _timerSim.WaitAsync(5);
			END_IF
      
      Await(_timerSim, nextStep:=QualityInspectionStep.StopEnd);
      // _step.SetNext(index:=QualityInspectionStep.StopEnd);

    (* -------------------------------------------------------------------------------------------------------------------------------- *)
    QualityInspectionStep.StopEnd:
    (* -------------------------------------------------------------------------------------------------------------------------------- *)    
      SetBusy(FALSE);
  
  ELSE
    Abort('sequence contains unhandled step');
  END_CASE
UNTIL _step.IsNotRepeatable() OR_ELSE NOT Busy END_REPEAT

END_FUNCTION_BLOCK

// ---- ZApp/Unit/QualityInspection/_States/QualityInspectionSequenceGoHome.TcPOU
FUNCTION_BLOCK QualityInspectionSequenceGoHome EXTENDS QualityInspectionSequence IMPLEMENTS ZCore.ISequence
VAR
  _step : ZCore.Step(QualityInspectionStep.GohomeBegin, QualityInspectionStep.GohomeEnd);
  _timer : ZAux.Timer;
END_VAR

IF NOT Busy THEN
  RETURN;
END_IF

IF OnStart(_step) THEN
  ; // init custom sequence variables here ...
END_IF

IF OnStop() THEN
  RETURN; // external stop was triggered
END_IF

IF OnHalt() THEN
  ; // Halting := TRUE; // Uncomment to acknowledge that the sequence is halting
END_IF

REPEAT
  LogStep();

  CASE _step.Index OF
    (* -------------------------------------------------------------------------------------------------------------------------------- *)
    QualityInspectionStep.GoHomeBegin:
    (* -------------------------------------------------------------------------------------------------------------------------------- *)
      IF _step.OnEntry()
      THEN
        _io.EnableLight.Enable(FALSE);
        _io.TriggerCam.Enable(FALSE);
        _timer.WaitAsync(1.0);
			END_IF
      
      Await(_timer, nextStep:=QualityInspectionStep.GoHomeEnd);

    (* -------------------------------------------------------------------------------------------------------------------------------- *)
    QualityInspectionStep.GoHomeEnd:
    (* -------------------------------------------------------------------------------------------------------------------------------- *)
      SetBusy(FALSE);
  
  ELSE
    Abort('sequence contains unhandled step');
  END_CASE
UNTIL _step.IsNotRepeatable() OR_ELSE NOT Busy END_REPEAT

END_FUNCTION_BLOCK

// ---- ZApp/Unit/QualityInspection/_States/QualityInspectionSequenceFaultReaction.TcPOU
FUNCTION_BLOCK QualityInspectionSequenceFaultReaction EXTENDS QualityInspectionSequence IMPLEMENTS ZCore.ISequence
VAR
  _step : ZCore.Step(QualityInspectionStep.FaultReactionBegin, QualityInspectionStep.FaultReactionEnd);
  _timerSim : ZAux.Timer;
END_VAR

IF OnStart(_step) THEN
  ; // init custom sequence variables here ...
END_IF

REPEAT
  LogStep();

  CASE _step.Index OF
    (* -------------------------------------------------------------------------------------------------------------------------------- *)
    QualityInspectionStep.FaultReactionBegin:
    (* -------------------------------------------------------------------------------------------------------------------------------- *)
      IF _step.OnEntry()
      THEN
        _timerSim.WaitAsync(5);
			END_IF
      
      Await(_timerSim, nextStep:=QualityInspectionStep.FaultReactionEnd);
      // _step.SetNext(index:=QualityInspectionStep.FaultReactionEnd);

    (* -------------------------------------------------------------------------------------------------------------------------------- *)
    QualityInspectionStep.FaultReactionEnd:
    (* -------------------------------------------------------------------------------------------------------------------------------- *)    
      SetBusy(FALSE);
  
  ELSE
    Abort('sequence contains unhandled step');
  END_CASE
UNTIL _step.IsNotRepeatable() OR_ELSE NOT Busy END_REPEAT

END_FUNCTION_BLOCK

// ---- ZApp/Unit/Assembly/AssemblyUnitProgram.TcPOU
/// each unit can run in its own PROGRAM and Task, respectively. However, this is optional and one may also
/// instantiate the unit in the ModuleProgram.
/// In order to keep initialization to a minimum, all ModuleContext objects that are required by the Unit are
/// given as FB_init parameter. These objects are
/// * data structs
/// * communication structs
/// * busmaster(s)
/// A unit should always be a root object (no parent) if it is running in its own context. If it runs in the same
/// task as the Module the parent may be set to the Module's Application.
PROGRAM AssemblyUnitProgram
VAR
{region "Assembly"}
{undefine RunInSeparateProgram}
{IF NOT (defined (Assembly_disabled)) AND (defined (RunInSeparateProgram))}
  Assembly : AssemblyUnit(name := 'Assembly', // name of the unit (for logging)
					  parent := 0, // caller of the Unit's cyclic method. If the Unit runs in its own context use 0
						configdata := ZGlobal.Data.Config.Assembly,
						machinedata := ZGlobal.Data.Machine.Assembly,
						calibrationdata := ZGlobal.Data.Calibration.Assembly,
						com := ZGlobal.Com.Unit.Assembly);
  {attribute 'section' := '__ZwPlcUnitProgramDeclaration__'}
  {attribute 'ZId' := 'fe48c71e-df5c-4f02-81a6-6f01ddca37c0'}
{END_IF}
{endregion}
{attribute '__ZwPlcUnitProgramDeclaration__'} // Do not remove this attribute! It is used for code generation.
END_VAR

// run the unit - the cylics of all children will be called as well

{region "Assembly"}
{undefine RunInSeparateProgram}
{IF NOT (defined (Assembly_disabled)) AND (defined (RunInSeparateProgram))}
  Assembly.Cyclic();
  {attribute 'section' := '__ZwPlcUnitProgramImplementation__'}
  {attribute 'ZId' := 'fe48c71e-df5c-4f02-81a6-6f01ddca37c0'}
{END_IF}
{endregion}
{attribute '__ZwPlcUnitProgramImplementation__'} // Do not remove this attribute! It is used for code generation.

END_PROGRAM

// ---- ZApp/Unit/Drilling/DrillingUnitProgram.TcPOU
/// each unit can run in its own PROGRAM and Task, respectively. However, this is optional and one may also
/// instantiate the unit in the ModuleProgram.
/// In order to keep initialization to a minimum, all ModuleContext objects that are required by the Unit are
/// given as FB_init parameter. These objects are
/// * data structs
/// * communication structs
/// * busmaster(s)
/// A unit should always be a root object (no parent) if it is running in its own context. If it runs in the same
/// task as the Module the parent may be set to the Module's Application.
PROGRAM DrillingUnitProgram
VAR
{region "Drilling"}
{undefine RunInSeparateProgram}
{IF NOT (defined (Drilling_disabled)) AND (defined (RunInSeparateProgram))}
  Drilling : DrillingUnit(name := 'Drilling', // name of the unit (for logging)
					  parent := 0, // caller of the Unit's cyclic method. If the Unit runs in its own context use 0
						configdata := ZGlobal.Data.Config.Drilling,
						machinedata := ZGlobal.Data.Machine.Drilling,
						calibrationdata := ZGlobal.Data.Calibration.Drilling,
						com := ZGlobal.Com.Unit.Drilling);
  {attribute 'section' := '__ZwPlcUnitProgramDeclaration__'}
  {attribute 'ZId' := 'a0f6f6d1-15cf-44f1-8585-ff8bdaab6c0e'}
{END_IF}
{endregion}
{attribute '__ZwPlcUnitProgramDeclaration__'} // Do not remove this attribute! It is used for code generation.
END_VAR

// run the unit - the cylics of all children will be called as well

{region "Drilling"}
{undefine RunInSeparateProgram}
{IF NOT (defined (Drilling_disabled)) AND (defined (RunInSeparateProgram))}
  Drilling.Cyclic();
  {attribute 'section' := '__ZwPlcUnitProgramImplementation__'}
  {attribute 'ZId' := 'a0f6f6d1-15cf-44f1-8585-ff8bdaab6c0e'}
{END_IF}
{endregion}
{attribute '__ZwPlcUnitProgramImplementation__'} // Do not remove this attribute! It is used for code generation.

END_PROGRAM

// ---- ZApp/Unit/QualityInspection/QualityInspectionUnitProgram.TcPOU
/// each unit can run in its own PROGRAM and Task, respectively. However, this is optional and one may also
/// instantiate the unit in the ModuleProgram.
/// In order to keep initialization to a minimum, all ModuleContext objects that are required by the Unit are
/// given as FB_init parameter. These objects are
/// * data structs
/// * communication structs
/// * busmaster(s)
/// A unit should always be a root object (no parent) if it is running in its own context. If it runs in the same
/// task as the Module the parent may be set to the Module's Application.
PROGRAM QualityInspectionUnitProgram
VAR
{region "QualityInspection"}
{undefine RunInSeparateProgram}
{IF NOT (defined (QualityInspection_disabled)) AND (defined (RunInSeparateProgram))}
  QualityInspection : QualityInspectionUnit(name := 'QualityInspection', // name of the unit (for logging)
					  parent := 0, // caller of the Unit's cyclic method. If the Unit runs in its own context use 0
						configdata := ZGlobal.Data.Config.QualityInspection,
						machinedata := ZGlobal.Data.Machine.QualityInspection,
						calibrationdata := ZGlobal.Data.Calibration.QualityInspection,
						com := ZGlobal.Com.Unit.QualityInspection);
  {attribute 'section' := '__ZwPlcUnitProgramDeclaration__'}
  {attribute 'ZId' := 'a1721ee9-e163-4dba-818e-d45d6db51cc5'}
{END_IF}
{endregion}
{attribute '__ZwPlcUnitProgramDeclaration__'} // Do not remove this attribute! It is used for code generation.
END_VAR

// run the unit - the cylics of all children will be called as well

{region "QualityInspection"}
{undefine RunInSeparateProgram}
{IF NOT (defined (QualityInspection_disabled)) AND (defined (RunInSeparateProgram))}
  QualityInspection.Cyclic();
  {attribute 'section' := '__ZwPlcUnitProgramImplementation__'}
  {attribute 'ZId' := 'a1721ee9-e163-4dba-818e-d45d6db51cc5'}
{END_IF}
{endregion}
{attribute '__ZwPlcUnitProgramImplementation__'} // Do not remove this attribute! It is used for code generation.

END_PROGRAM

// ---- ZApp/Unit/Transport/TransportUnitProgram.TcPOU
/// each unit can run in its own PROGRAM and Task, respectively. However, this is optional and one may also
/// instantiate the unit in the ModuleProgram.
/// In order to keep initialization to a minimum, all ModuleContext objects that are required by the Unit are
/// given as FB_init parameter. These objects are
/// * data structs
/// * communication structs
/// * busmaster(s)
/// A unit should always be a root object (no parent) if it is running in its own context. If it runs in the same
/// task as the Module the parent may be set to the Module's Application.
PROGRAM TransportUnitProgram
VAR
{region "Transport"}
{undefine RunInSeparateProgram}
{IF NOT (defined (Transport_disabled)) AND (defined (RunInSeparateProgram))}
  Transport : TransportUnit(name := 'Transport', // name of the unit (for logging)
					  parent := 0, // caller of the Unit's cyclic method. If the Unit runs in its own context use 0
						configdata := ZGlobal.Data.Config.Transport,
						machinedata := ZGlobal.Data.Machine.Transport,
						calibrationdata := ZGlobal.Data.Calibration.Transport,
						com := ZGlobal.Com.Unit.Transport);
  {attribute 'section' := '__ZwPlcUnitProgramDeclaration__'}
  {attribute 'ZId' := '413070d6-61de-4759-aae5-e3ab76278fe1'}
{END_IF}
{endregion}
{attribute '__ZwPlcUnitProgramDeclaration__'} // Do not remove this attribute! It is used for code generation.
END_VAR

// run the unit - the cylics of all children will be called as well

{region "Transport"}
{undefine RunInSeparateProgram}
{IF NOT (defined (Transport_disabled)) AND (defined (RunInSeparateProgram))}
  Transport.Cyclic();
  {attribute 'section' := '__ZwPlcUnitProgramImplementation__'}
  {attribute 'ZId' := '413070d6-61de-4759-aae5-e3ab76278fe1'}
{END_IF}
{endregion}
{attribute '__ZwPlcUnitProgramImplementation__'} // Do not remove this attribute! It is used for code generation.

END_PROGRAM
